TYPE T_Ctrl_SIf_STB_Cur :
STRUCT
	/// Hangers passed total counter (reset in state OFF)
	dinHangersPassedTotal: DINT;
	/// Hangers passed package counter (is updated when “RELEASE_ALL” command is completed)
	dinHangersPassedPackage: DINT;
	/// Hanger detected
	bolHangerDetected: BOOL;
	/// Approximate number of hangers in buffer
	dinNumOfHangersInBuffer: DINT;
	/// Buffer is full
	bolBufferFull: BOOL;
	/// Pointer to section buffer of FUB MTR. Needed in case if STB work in combination with MTR to merge hangers into a TLK.
	pSectionBuffer: POINTER TO ARRAY[0..Const_MTR.cusiSectionBuffer_SIZE] OF T_MTR_Buffer_Sections;
	///[um] actual position from the transport written from Parent
	dinTransportPosition_um: DINT;
	///[um] actual speed from the transport written from Parent
	dinTransportspeed_um_s: DINT;
	///[um] actual calculated position
	dinTransportPositionCalc_um: DINT;
END_STRUCT
END_TYPE

(* stored: Version 1.1.0.1, ProductVersion 3.1.0.23
   DUT T_Ctrl_SIf_STB_Cur: Id {2ba6579a-d993-45fc-b27e-22669bb1d6e4} *)
